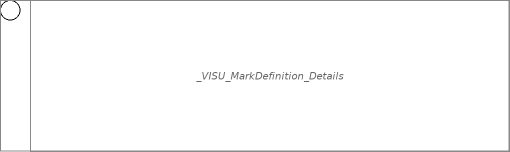
VISUALIZATION _VISU_MarkDefinition  // 510x152
VAR_IN_OUT
	mInst : FB_MarkDefinition;
END_VAR
    Ellipse (0,0 20x20), tooltip "Mark Details"
        toggle mInst.bShowDetail
    Frame (30,0 480x152), invisible if: NOT mInst.bShowDetail
        shows _VISU_MarkDefinition_Details(mInst := mInst)
END_VISUALIZATION

(* stored: Version 1.1.0.1, ProductVersion 3.1.4024.11
   Visu _VISU_MarkDefinition: Id {1e1151fd-e3e6-4c3b-8ab8-f03914dc3a32} *)
